(* PLC project Generated.project, CODESYS CODESYS V3.5 SP19 Patch 1 *)
(* stored: creationDateTime 2026-08-27T17:21:57.492816, modificationDateTime 2026-08-27T17:21:57.492816 *)

(* ======================================================================= ⚙️ ST_fbEncoder_Cfg — Réglages technologiques publics de FB_Encoder ─────────────────────────────────────────────────────────────────────── 🎯 Rôle : porter le mode de confirmation preset commun aux codeurs. 🔒 Ownership : GVL_IHM.Commun.EncoderCfg ↔ GVL_PERSISTENT._EncoderCfgPersist. 📄 Doc : DOC/AF/AF_Partie-09_Fonction_Encoder_v2.3.md ======================================================================= *)
TYPE ST_fbEncoder_Cfg : STRUCT
  PresetConfirmMode : E_PresetConfirmMode := E_PresetConfirmMode.READBACK_ONLY;  (* Mode de confirmation preset, défaut relecture *)
  Initialized : BOOL := FALSE;  (* 🚦 TRUE après restauration du pont persistant *)
END_STRUCT;
END_TYPE

(* values of E_PresetConfirmMode: READBACK_ONLY: Confirmation par relecture de position; READBACK_AND_STATUSBIT: Relecture et bit d'état matériel; STATUSBIT_ONLY: Bit d'état matériel uniquement *)

{attribute 'qualified_only'}
{attribute 'strict'}
TYPE E_PresetConfirmMode : (READBACK_ONLY := 0, READBACK_AND_STATUSBIT := 1, STATUSBIT_ONLY := 2);
END_TYPE
